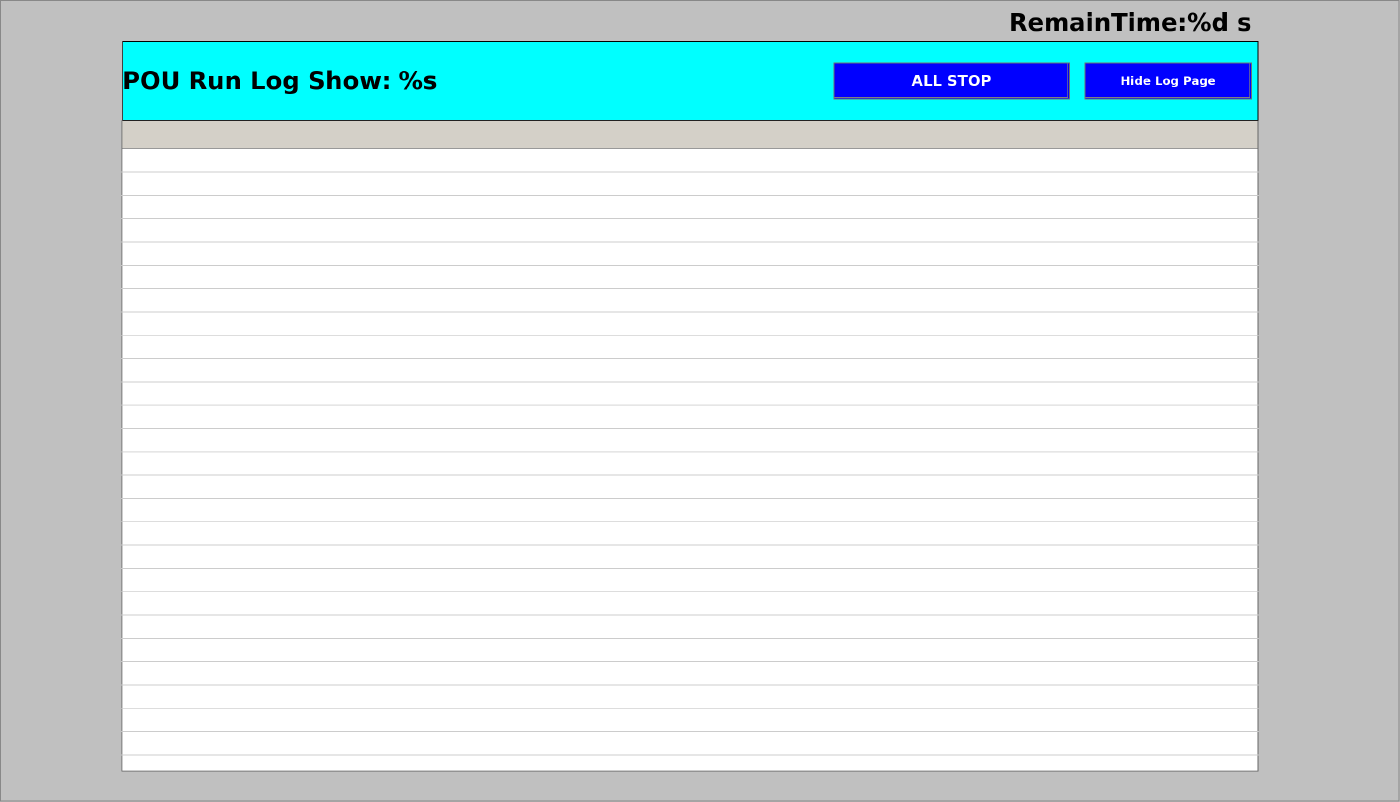
VISUALIZATION showInfo_Auto  // 1500x860
VAR_IN_OUT
	userData: printLogModule_EX_DataHMI;
END_VAR
    Rectangle (0,0 1500x860)
    Table (130,129 1218x698), data array: userData.logStrData
        p1128707560: cNumLength_showInof
        p3854506369: userData.logStrData[INDEX].sTime
        p1892666644: userData.logStrData[INDEX].msg
        p511219082: Information
    RoundedRectangle (131,44 1217x85)
    Label (133,57 285x59), "POU Run Log Show:"
    Button (1162,67 179x39), "Hide Log Page"
        OnMouseClick: execute { gShowPOURunLog:=NOT gShowPOURunLog; }
    Button (893,67 253x39), "ALL STOP"
        tap MainRunPOU.AllAbort
        OnMouseClick: execute {
            gShowPOURunLog:=NOT gShowPOURunLog;
            gCtrlMode:=ControlMode.eManualCtrMode;
            IF RunningStatus.eErrorState<>gRunningState THEN
            	gRunningState:=RunningStatus.eManualState;
            END_IF
        }
    Rectangle (424,51 443x71), "%s", text variable: gShowLogTextTitle
    Rectangle (1003,3 341x42), "RemainTime:%d s", text variable: gCO_ControlRFRMTime, invisible if: NOT S_CO_ControlRF.busy
END_VISUALIZATION

(* stored: Version 1.1.0.1, ProductVersion 3.1.4024.12
   Visu showInfo_Auto: Id {2f486119-1b4b-439a-81ff-108da0666e84} *)
